PROGRAM Motion
VAR
	/// axis reference data structure 
	Axis1: AXIS_REF;
	/// state machine state 
	state: MoveState_t;
	PowerAxis1: MC_Power;
	/// debug function block output data 
	PowerAxis1Out: ST_McOutputs;
	MoveAxis1: MC_MoveAbsolute;
	/// debug function block output data 
	MoveAbsoluteOut1: ST_McOutputs;
	MoveAxis2: MC_MoveAbsolute;
	/// debug function block output data 
	MoveAbsoluteOut2: ST_McOutputs;
	Reset: MC_Reset;
	/// debug function block output data 
	ResetOut: ST_McOutputs;
	
	autoOut		: F_TRIG;
END_VAR

(* update the axis status at the beginning of each cycle *)
Axis1();

autoOut(CLK:=GVL.bRunning);
IF autoOut.Q THEN
	state := MOVESTATE_RESET;
END_IF

(* move axis using a state machine *)
CASE state OF

	MOVESTATE_INIT :	(* initialisation *)
		(* initialize all function blocks *)
		MoveAxis1.Execute := FALSE;
		MoveAxis2.Execute := FALSE;
		Reset.Execute := FALSE;
		state := MOVESTATE_ENABLE;

	MOVESTATE_ENABLE :
		PowerAxis1.Enable := TRUE;
		PowerAxis1.Enable_Positive := TRUE;
		PowerAxis1.Enable_Negative := TRUE;
		IF PowerAxis1.Status THEN
			IF GVL.bRunning THEN
				state := MOVESTATE_FORWARD;
			END_IF
		ELSIF PowerAxis1.Error THEN
			state := MOVESTATE_ERROR;
		END_IF

	MOVESTATE_FORWARD :		(* start to first position *)
		MoveAxis1.Position := 1500;		(* start to intermediate tartet position *)
		MoveAxis1.Velocity := 500;		(* medium velocity level *)
		MoveAxis1.BufferMode := MC_Buffered;
		MoveAxis1.Execute := TRUE;
		IF MoveAxis1.Active  THEN
			(* axis is executing job but is not yet finished *)
			MoveAxis1.Execute := FALSE;
			(* leave this state and buffer a second command *)
			state := MOVESTATE_NEWTARGETPOSITION;
		ELSIF MoveAxis1.CommandAborted OR MoveAxis1.Error THEN
			state := MOVESTATE_ERROR;
		END_IF

	MOVESTATE_NEWTARGETPOSITION :		(* change target position while moving *)
		(* start a buffered motion command while axis is moving *)
		MoveAxis2.Position := 5000;		(* start to final target *)
		MoveAxis2.Velocity := 1500;		(* increase velocity *)
		MoveAxis2.BufferMode := MC_BlendingPrevious; 	(* use velocity of previous command till intermediate target position position *)
		MoveAxis2.Execute := TRUE;
		IF MoveAxis2.Done THEN
			MoveAxis2.Execute := FALSE;
			state := MOVESTATE_BACKWARDS;
		ELSIF MoveAxis2.CommandAborted OR MoveAxis2.Error THEN
			state := MOVESTATE_ERROR;
		END_IF

	MOVESTATE_BACKWARDS :	(* move back to initial position *)
		MoveAxis1.Position := 100;		(* position close to initial position *)
		MoveAxis1.Velocity := 2000;		(* high velocity *)
		MoveAxis1.BufferMode := MC_Buffered;
		MoveAxis1.Execute := TRUE;
		IF MoveAxis1.Active THEN
			(* axis is executing job but is not yet finished *)
			MoveAxis1.Execute := FALSE;
			(* leave this state and buffer a second command *)
			state := MOVESTATE_BACKWARDSSLOW;
		ELSIF MoveAxis1.CommandAborted OR MoveAxis1.Error THEN
			state := MOVESTATE_ERROR;
		END_IF

	MOVESTATE_BACKWARDSSLOW :	(* move back to initial position *)
		(* start a buffered motion command while axis is moving *)
		MoveAxis2.Position := 0;	(* back to initial position *)
		MoveAxis2.Velocity := 100; 	(* slow velocity *)
		MoveAxis2.BufferMode := MC_BlendingNext; 	(* use velocity from first target position *)
		MoveAxis2.Execute := TRUE;
		IF MoveAxis2.Done THEN
			MoveAxis2.Execute := FALSE;
			state := MOVESTATE_FORWARD;
		ELSIF MoveAxis2.CommandAborted OR MoveAxis2.Error THEN
			state := MOVESTATE_ERROR;
		END_IF

	MOVESTATE_ERROR :
		IF Axis1.Status.Error THEN
			state := MOVESTATE_RESET;	(* axis error requires reset *)
		ELSE
			state := MOVESTATE_INIT;		(* function block errors don't need a reset *)
		END_IF

	MOVESTATE_RESET :
		Reset.Execute := TRUE;
		IF Reset.Done THEN
			state := MOVESTATE_INIT;
		ELSIF Reset.Error THEN
			state := MOVESTATE_INIT; (* can't do anything here *)
		END_IF

END_CASE

ActPower();	(* call the power function block *)
ActMove();	(* call the move function block *)
ActReset();	(* call the reset function block *)

ACTION ActMove:
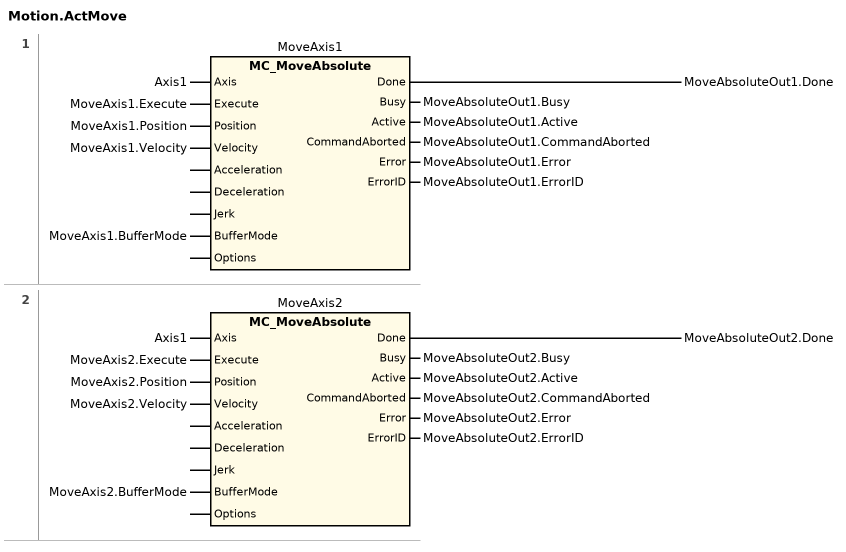
// NETWORK 1
MoveAxis1(
    Axis := Axis1,
    Execute := MoveAxis1.Execute,
    Position := MoveAxis1.Position,
    Velocity := MoveAxis1.Velocity,
    BufferMode := MoveAxis1.BufferMode,
    Busy => MoveAbsoluteOut1.Busy,
    Active => MoveAbsoluteOut1.Active,
    CommandAborted => MoveAbsoluteOut1.CommandAborted,
    Error => MoveAbsoluteOut1.Error,
    ErrorID => MoveAbsoluteOut1.ErrorID); // MC_MoveAbsolute
MoveAbsoluteOut1.Done := MoveAxis1.Done;

// NETWORK 2
MoveAxis2(
    Axis := Axis1,
    Execute := MoveAxis2.Execute,
    Position := MoveAxis2.Position,
    Velocity := MoveAxis2.Velocity,
    BufferMode := MoveAxis2.BufferMode,
    Busy => MoveAbsoluteOut2.Busy,
    Active => MoveAbsoluteOut2.Active,
    CommandAborted => MoveAbsoluteOut2.CommandAborted,
    Error => MoveAbsoluteOut2.Error,
    ErrorID => MoveAbsoluteOut2.ErrorID); // MC_MoveAbsolute
MoveAbsoluteOut2.Done := MoveAxis2.Done;
END_ACTION

ACTION ActPower:
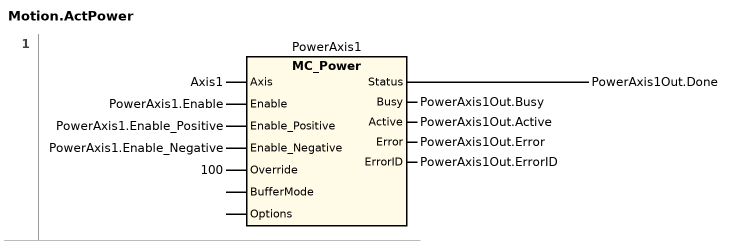
// NETWORK 1
PowerAxis1(
    Axis := Axis1,
    Enable := PowerAxis1.Enable,
    Enable_Positive := PowerAxis1.Enable_Positive,
    Enable_Negative := PowerAxis1.Enable_Negative,
    Override := 100,
    Busy => PowerAxis1Out.Busy,
    Active => PowerAxis1Out.Active,
    Error => PowerAxis1Out.Error,
    ErrorID => PowerAxis1Out.ErrorID); // MC_Power
PowerAxis1Out.Done := PowerAxis1.Status;
END_ACTION

ACTION ActReset:
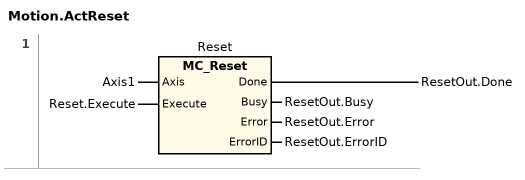
// NETWORK 1
Reset(
    Axis := Axis1,
    Execute := Reset.Execute,
    Busy => ResetOut.Busy,
    Error => ResetOut.Error,
    ErrorID => ResetOut.ErrorID); // MC_Reset
ResetOut.Done := Reset.Done;
END_ACTION

END_PROGRAM

(* stored: Version 1.1.0.1
   POU Motion: Id {3a666bc5-dba5-4381-89e8-d29bc58c73bc}, SpecialFunc None
   Action ActMove: Id {795d9605-c228-45e1-99c5-4ec8f5706771}
   Action ActPower: Id {6f998a64-4472-46bb-acb0-ad84cdb6ed24}
   Action ActReset: Id {8f6bb17b-609e-4e92-b12c-1c5d1a94aec2} *)
